FUNCTION_BLOCK F_CONCAT_2 (* concatenation of two strings *)
  (* Standard: 61131-3; Classification: standard character and string function; Description: Copyright (c) 2013 TU Wien ACIN, HR Agrartechnik GmbH This program and the accompanying materials are made available under the terms of the Eclipse Public License 2.0 which is available at https://www.eclipse.org/legal/epl-2.0/ SPDX-License-Identifier: EPL-2.0 *)
  (* Version 1.0, 2026-02-01, Franz Höpfinger, HR Agrartechnik GmbH, Copy over from F_CONCAT and made this Block *)
  PACKAGE iec61131::charString;
  {SET_ATTRIBUTE(eclipse4diac::core::GenericClassName, 'GEN_CONCAT')}
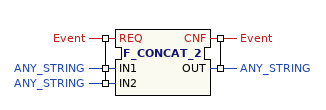
  EVENT_INPUT
    REQ WITH IN1, IN2; (* Service Request *)
  END_EVENT
  EVENT_OUTPUT
    CNF WITH OUT; (* Confirmation of Requested Service *)
  END_EVENT
  VAR_INPUT
    IN1 : ANY_STRING; (* input string 1 *)
    IN2 : ANY_STRING; (* input string 2 *)
  END_VAR
  VAR_OUTPUT
    OUT : ANY_STRING; (* Result *)
  END_VAR
END_FUNCTION_BLOCK
